FUNCTION_BLOCK FB_BarcodeScanner EXTENDS FB_Station
VAR_INPUT
END_VAR
VAR_OUTPUT
END_VAR
VAR
	bTriggerRead			AT %Q* : BOOL;
	sBarcode				AT %I* : STRING(255);
	
	sBarcodeRead			: STRING(255);
	iWorkState				: DINT;
	iRetries				: DINT;
	tmrRetry				: TON;
END_VAR
VAR CONSTANT
	NO_READ					: STRING(255) := 'NO_READ';
	READ_RETRY_COUNT		: DINT := 3;
END_VAR

METHOD PROTECTED  DoWork : BOOL
VAR_INPUT
END_VAR
CASE iWorkState OF
	0:
		iRetries := 0;
		sBarcodeRead := '';
		iWorkState := 10;
		bTriggerRead := TRUE;
		
	10:
		IF sBarcode <> '' THEN
			sBarcodeRead := sBarcode;
			bTriggerRead := FALSE;
			iWorkState := 20;
		END_IF
		
	11:
		tmrRetry(IN:=TRUE, PT:=T#500MS);
		IF tmrRetry.Q THEN
			tmrRetry(IN:=FALSE);
			bTriggerRead := TRUE;
			iWorkState := 20;
		END_IF
		
	20:
		IF sBarcodeRead = NO_READ THEN
			IF iRetries < READ_RETRY_COUNT THEN
				iRetries := iRetries + 1;
				iWorkState := 11;
			ELSE
				pPartStatus^.bBarcodeStatus := FALSE;
				pPartStatus^.sBarcode := NO_READ;
				iWorkState := 30;
			END_IF
		ELSE
			pPartStatus^.bBarcodeStatus := TRUE;
			pPartStatus^.sBarcode := sBarcodeRead;
			iWorkState := 30;
		END_IF
		
	30:
		iWorkState := 0;
		DoWork := TRUE;
	
END_CASE
END_METHOD

METHOD PROTECTED  FaultHandler : E_StationState
VAR_INPUT
END_VAR
END_METHOD

END_FUNCTION_BLOCK

(* stored: Version 1.1.0.1, ProductVersion 3.1.4024.12
   POU FB_BarcodeScanner: Id {83862807-4f6b-4b20-89ce-4ca729399ad6}, SpecialFunc None
   Method DoWork: Id {d51b3fb6-d4ff-4009-ab0d-2fab363dee34}
   Method FaultHandler: Id {54f9818e-7814-4bbf-b316-1b6a174d9bf6} *)
